(* PLC project desalination, Generated TextualNotationConverter 1.0 *)
(* stored: creationDateTime 2025-07-30T12:00:00, modificationDateTime 2025-01-30T12:00:00 *)

FUNCTION_BLOCK ANALOG_IN
  VAR_INPUT
    Name : STRING;
    Description : STRING;
    Raw_Signal : REAL;
    PV_High : REAL;
    PV_Low : REAL;
    Scaling_Slope : REAL;
    Scaling_Offset : REAL;
    Alarm_Enable : BOOL;
  END_VAR
  VAR_OUTPUT
    PV : REAL;
    High_Alarm : BOOL;
    Low_Alarm : BOOL;
    General_Fault : BOOL;
  END_VAR

            
          
END_FUNCTION_BLOCK

FUNCTION_BLOCK DIGITAL_IN
  VAR_INPUT
    Name : STRING;
    Description : STRING;
    DI_Raw : BOOL;
    DebounceTime : STRING;
    EnableAlarm : BOOL;
  END_VAR
  VAR_OUTPUT
    DI_Out : BOOL;
    Fault_State : BOOL;
  END_VAR

            
          
END_FUNCTION_BLOCK

FUNCTION_BLOCK PID_BASIC
  VAR_INPUT
    Name : STRING;
    Description : STRING;
    AUTO : BOOL;
    PV : REAL;
    SP : REAL;
    MV_MIN : REAL;
    MV_MAX : REAL;
    X0 : REAL;
    KP : REAL;
    TR : REAL;
    TD : REAL;
    PV_High : REAL;
    PV_Low : REAL;
    Deviation_Limit : REAL;
    Inhibit : BOOL;
  END_VAR
  VAR_OUTPUT
    PV_High_Alarm : BOOL;
    PV_Low_Alarm : BOOL;
    Deviation_Alarm : BOOL;
    XOUT : REAL;
  END_VAR

            
          
END_FUNCTION_BLOCK

FUNCTION_BLOCK VALVE_ELECTRIC
  VAR_INPUT
    Name : STRING;
    Description : STRING;
    Control_Signal : REAL;
    Manual_Mode : BOOL;
    Manual_Position : REAL;
    Open_Limit : REAL;
    Close_Limit : REAL;
    Timeout : STRING;
    Inhibit : BOOL;
  END_VAR
  VAR_OUTPUT
    Valve_Position : REAL;
    Feedback_Pos : REAL;
    Valve_Moving : BOOL;
    Position_Error : BOOL;
    Alarm : BOOL;
  END_VAR

            
          
END_FUNCTION_BLOCK

FUNCTION_BLOCK VALVE_ON_OFF
  VAR_INPUT
    Name : STRING;
    Description : STRING;
    Open_Cmd : BOOL;
    Close_Cmd : BOOL;
    Timeout : STRING;
    Inhibit : BOOL;
  END_VAR
  VAR_OUTPUT
    FB_Opened : BOOL;
    FB_Closed : BOOL;
    Valve_Open_Out : BOOL;
    Valve_Close_Out : BOOL;
    Alarm_Position_Error : BOOL;
    Alarm_General : BOOL;
  END_VAR

            
          
END_FUNCTION_BLOCK

PROGRAM Section2
  VAR
    AT_101_mA : REAL;
    AT_103_mA : REAL;
    FT_101_mA : REAL;
    FT_102_mA : REAL;
    LT_104_mA : REAL;
    LT_105_mA : REAL;
    XV_102_OpenLS_Raw : BOOL;
    XV_102_CloseLS_Raw : BOOL;
    SP_Seawater_Req : REAL;
    SP_Reservoir_Req : REAL;
    SP_Seawater_Clamped : REAL;
    SP_Reservoir_Clamped : REAL;
    FC_101_Auto_Cmd : BOOL;
    FC_102_Auto_Cmd : BOOL;
    FV_101_Manual_Mode : BOOL;
    FV_102_Manual_Mode : BOOL;
    FV_101_Manual_Position : REAL;
    FV_102_Manual_Position : REAL;
    FT_101_Flow_PV : REAL;
    FT_102_Flow_PV : REAL;
    FC_101_PID_Output : REAL;
    FC_102_PID_Output : REAL;
    FV_101_Valve_Position : REAL;
    FV_102_Valve_Position : REAL;
    AT_101_Quality_PV : REAL;
    AT_103_Quality_PV : REAL;
    LT_104_Level_PV : REAL;
    LT_105_Level_PV : REAL;
    WaterQuality_Alarm : BOOL;
    FV101_Inhibit : BOOL;
    FV102_Inhibit : BOOL;
  END_VAR
  VAR
    AT-101 : ANALOG_IN;
    AT-103 : ANALOG_IN;
    FC-101 : PID_BASIC;
    FC-102 : PID_BASIC;
    FT-101 : ANALOG_IN;
    FT-102 : ANALOG_IN;
    FV-101 : VALVE_ELECTRIC;
    FV-102 : VALVE_ELECTRIC;
    LT-104 : ANALOG_IN;
    LT-105 : ANALOG_IN;
    XV-102 : VALVE_ON_OFF;
    XV-102_OPEN_LS : DIGITAL_IN;
    XV-102_CLOSE_LS : DIGITAL_IN;
  END_VAR
  VAR  (* added by the conversion: wires and edge detectors of the diagram *)
    _OR1_OUT : BOOL;
    _OR2_OUT : BOOL;
    _OR3_OUT : BOOL;
  END_VAR

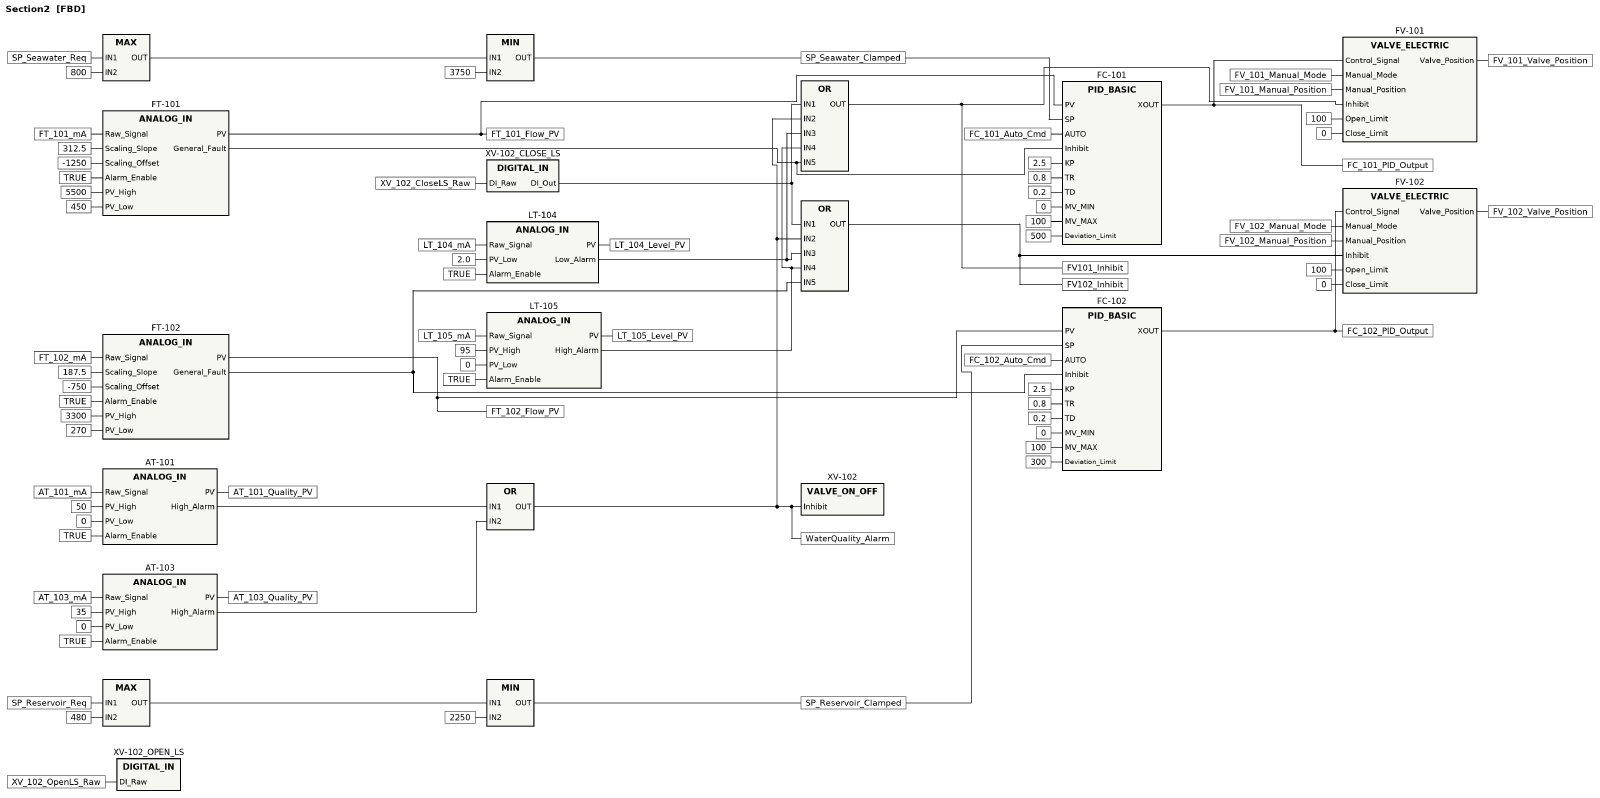
(* FBD diagram, written out as Structured Text *)
AT-101(Raw_Signal := AT_101_mA, PV_High := 50, PV_Low := 0, Alarm_Enable := TRUE);
AT_101_Quality_PV := AT-101.PV;
AT-103(Raw_Signal := AT_103_mA, PV_High := 35, PV_Low := 0, Alarm_Enable := TRUE);
AT_103_Quality_PV := AT-103.PV;
FT-101(Raw_Signal := FT_101_mA, Scaling_Slope := 312.5, Scaling_Offset := -1250, Alarm_Enable := TRUE, PV_High := 5500, PV_Low := 450);
FC-101(PV := FT-101.PV, SP := MIN(MAX(SP_Seawater_Req, 800), 3750), AUTO := FC_101_Auto_Cmd, Inhibit := FT-101.General_Fault, KP := 2.5, TR := 0.8, TD := 0.2, MV_MIN := 0, MV_MAX := 100, Deviation_Limit := 500);
FC_101_PID_Output := FC-101.XOUT;
FT-102(Raw_Signal := FT_102_mA, Scaling_Slope := 187.5, Scaling_Offset := -750, Alarm_Enable := TRUE, PV_High := 3300, PV_Low := 270);
FC-102(PV := FT-102.PV, SP := MIN(MAX(SP_Reservoir_Req, 480), 2250), AUTO := FC_102_Auto_Cmd, Inhibit := FT-102.General_Fault, KP := 2.5, TR := 0.8, TD := 0.2, MV_MIN := 0, MV_MAX := 100, Deviation_Limit := 300);
FC_102_PID_Output := FC-102.XOUT;
FT_101_Flow_PV := FT-101.PV;
FT_102_Flow_PV := FT-102.PV;
XV-102_CLOSE_LS(DI_Raw := XV_102_CloseLS_Raw);
_OR1_OUT := AT-101.High_Alarm OR AT-103.High_Alarm;
LT-104(Raw_Signal := LT_104_mA, PV_Low := 2.0, Alarm_Enable := TRUE);
LT-105(Raw_Signal := LT_105_mA, PV_High := 95, PV_Low := 0, Alarm_Enable := TRUE);
_OR2_OUT := XV-102_CLOSE_LS.DI_Out OR _OR1_OUT OR LT-104.Low_Alarm OR LT-105.High_Alarm OR FT-101.General_Fault;
FV101_Inhibit := _OR2_OUT;
_OR3_OUT := XV-102_CLOSE_LS.DI_Out OR _OR1_OUT OR LT-104.Low_Alarm OR LT-105.High_Alarm OR FT-102.General_Fault;
FV102_Inhibit := _OR3_OUT;
FV-101(Control_Signal := FC-101.XOUT, Manual_Mode := FV_101_Manual_Mode, Manual_Position := FV_101_Manual_Position, Inhibit := _OR2_OUT, Open_Limit := 100, Close_Limit := 0);
FV_101_Valve_Position := FV-101.Valve_Position;
FV-102(Control_Signal := FC-102.XOUT, Manual_Mode := FV_102_Manual_Mode, Manual_Position := FV_102_Manual_Position, Inhibit := _OR3_OUT, Open_Limit := 100, Close_Limit := 0);
FV_102_Valve_Position := FV-102.Valve_Position;
LT_104_Level_PV := LT-104.PV;
LT_105_Level_PV := LT-105.PV;
SP_Reservoir_Clamped := MIN(MAX(SP_Reservoir_Req, 480), 2250);
SP_Seawater_Clamped := MIN(MAX(SP_Seawater_Req, 800), 3750);
WaterQuality_Alarm := _OR1_OUT;
XV-102(Inhibit := _OR1_OUT);
XV-102_OPEN_LS(DI_Raw := XV_102_OpenLS_Raw);
END_PROGRAM

FUNCTION_BLOCK BOOL_IN
  VAR_INPUT
    Name : STRING;
    Description : STRING;
    Bool_In : BOOL;
    Alarm_OnTrue : BOOL;
    Alarm_OnFalse : BOOL;
    Latch_Enable : BOOL;
    Reset_Latch : BOOL;
  END_VAR
  VAR_OUTPUT
    Bool_Out : BOOL;
    Alarm_Active : BOOL;
    Latched_Status : BOOL;
  END_VAR

            
          
END_FUNCTION_BLOCK

FUNCTION_BLOCK DUTY_STANDBY
  VAR_INPUT
    Name : STRING;
    Description : STRING;
    Enable : BOOL;
    StartRequest : BOOL;
    AlternateEnable : BOOL;
    ForcePumpA : BOOL;
    ForcePumpB : BOOL;
    DutyElapsed : BOOL;
    MinRunElapsed : BOOL;
    SwitchoverDelayElapsed : BOOL;
    StartTimeoutElapsed : BOOL;
    PumpA_RunFB : BOOL;
    PumpB_RunFB : BOOL;
    PumpA_Fault : BOOL;
    PumpB_Fault : BOOL;
    Reset : BOOL;
    Inhibit : BOOL;
  END_VAR
  VAR_OUTPUT
    CmdPumpA : BOOL;
    CmdPumpB : BOOL;
    ActiveIsA : BOOL;
    SwitchedDueToDuty : BOOL;
    SwitchedDueToFailure : BOOL;
    Alarm_FailedStart_A : BOOL;
    Alarm_FailedStart_B : BOOL;
    Alarm_NoAvailablePump : BOOL;
  END_VAR

            
          
END_FUNCTION_BLOCK

FUNCTION_BLOCK MOTOR_2SPD
  VAR_INPUT
    Name : STRING;
    Description : STRING;
    Start_Cmd : BOOL;
    Stop_Cmd : BOOL;
    Speed_High_Cmd : BOOL;
    Speed_Low_Cmd : BOOL;
    Inhibit : BOOL;
  END_VAR
  VAR_OUTPUT
    Motor_Start_Out : BOOL;
    FB_Running : BOOL;
    FB_Trip : BOOL;
    FB_HighSpeed : BOOL;
    FB_LowSpeed : BOOL;
    Alarm_Speed_Error : BOOL;
  END_VAR

            
          
END_FUNCTION_BLOCK

FUNCTION_BLOCK MOTOR_ON_OFF
  VAR_INPUT
    Name : STRING;
    Description : STRING;
    Start_Cmd : BOOL;
    Stop_Cmd : BOOL;
    Start_Delay : STRING;
    MinRunTime : STRING;
    Inhibit : BOOL;
  END_VAR
  VAR_OUTPUT
    Motor_Start_Out : BOOL;
    FB_Running : BOOL;
    FB_Trip : BOOL;
    Alarm_Start_Fail : BOOL;
    Alarm_Stop_Fail : BOOL;
  END_VAR

            
          
END_FUNCTION_BLOCK

FUNCTION_BLOCK MOTOR_VSD
  VAR_INPUT
    Name : STRING;
    Description : STRING;
    Start_Cmd : BOOL;
    Stop_Cmd : BOOL;
    Speed_SP : REAL;
    Accel_Ramp : STRING;
    Decel_Ramp : STRING;
    Inhibit : BOOL;
  END_VAR
  VAR_OUTPUT
    Speed_Out : REAL;
    FB_Running : BOOL;
    FB_Fault : BOOL;
    FB_Ready : BOOL;
    FB_ActualSpeed : REAL;
    Alarm_Speed_Deviation : BOOL;
    Alarm_Comm_Fail : BOOL;
  END_VAR

            
          
END_FUNCTION_BLOCK

FUNCTION_BLOCK RATIO_CONTROL
  VAR_INPUT
    Name : STRING;
    Description : STRING;
    Auto : BOOL;
    PrimaryPV : REAL;
    SecondaryPV : REAL;
    RatioSP : REAL;
    Bias : REAL;
    TrimKp : REAL;
    TrimTi : STRING;
    MV_MIN : REAL;
    MV_MAX : REAL;
    ManOut : REAL;
    Inhibit : BOOL;
  END_VAR
  VAR_OUTPUT
    SlaveSP : REAL;
    ActiveRatio : REAL;
    RatioErr : REAL;
  END_VAR

            
          
END_FUNCTION_BLOCK

FUNCTION_BLOCK SPLIT_RANGE
  VAR_INPUT
    Name : STRING;
    Description : STRING;
    IN : REAL;
    Split_Point : REAL;
    Output1_Start : REAL;
    Output1_End : REAL;
    Output2_Start : REAL;
    Output2_End : REAL;
  END_VAR
  VAR_OUTPUT
    OUT1 : REAL;
    OUT2 : REAL;
  END_VAR

            
          
END_FUNCTION_BLOCK

FUNCTION_BLOCK VOTING_ANALOG
  VAR_INPUT
    Name : STRING;
    Description : STRING;
    Input1 : REAL;
    Input2 : REAL;
    Input3 : REAL;
    Deviation_Limit : REAL;
    Voting_Scheme : STRING;
    EnableAlarm : BOOL;
    Inhibit : BOOL;
  END_VAR
  VAR_OUTPUT
    Voted_Output : REAL;
    Sensor1_Fault : BOOL;
    Sensor2_Fault : BOOL;
    Sensor3_Fault : BOOL;
    Alarm_Voting_Error : BOOL;
    Healthy_Sensors_Count : INT;
  END_VAR

            
          
END_FUNCTION_BLOCK

PROGRAM Section3
  VAR
    FT101_SupplyAirFlow_PV : REAL;
    FT102_ScreenAirFlow_PV : REAL;
    PT103_UpstreamPressure_PV : REAL;
    PT104_DownstreamPressure_PV : REAL;
    PIT105_CompressedAirPressure_PV : REAL;
    PIT106_CleaningSystemPressure_PV : REAL;
    PT108_SupplyPressure_PV : REAL;
    FFIC103_SlaveSetpoint_FT102Flow : REAL;
    FIC104_ValveCommand_Percent : REAL;
    FV105_ValvePosition_Percent : REAL;
    FV105_FeedbackPosition_Percent : REAL;
    SW_SCREEN_1_Status : BOOL;
    SW_SCREEN_2_Status : BOOL;
    SW_SCREEN_3_Status : BOOL;
    SW_SCREEN_4_Status : BOOL;
    SW_SCREEN_5_Status : BOOL;
    SW_SCREEN_6_Status : BOOL;
    RES_SCREEN_1_Status : BOOL;
    RES_SCREEN_2_Status : BOOL;
    RES_SCREEN_3_Status : BOOL;
    RES_SCREEN_4_Status : BOOL;
  END_VAR
  VAR
    FFIC-103 : RATIO_CONTROL;
    FIC-104 : PID_BASIC;
    FV-105 : VALVE_ELECTRIC;
    FT-101 : ANALOG_IN;
    FT-102 : ANALOG_IN;
    PIT-105 : ANALOG_IN;
    PIT-106 : ANALOG_IN;
    PT-103 : ANALOG_IN;
    PT-104 : ANALOG_IN;
    PT-108 : ANALOG_IN;
    SW-SCREEN-1 : BOOL_IN;
    SW-SCREEN-2 : BOOL_IN;
    SW-SCREEN-3 : BOOL_IN;
    SW-SCREEN-4 : BOOL_IN;
    SW-SCREEN-5 : BOOL_IN;
    SW-SCREEN-6 : BOOL_IN;
    RES-SCREEN-1 : BOOL_IN;
    RES-SCREEN-2 : BOOL_IN;
    RES-SCREEN-3 : BOOL_IN;
    RES-SCREEN-4 : BOOL_IN;
  END_VAR
  VAR  (* added by the conversion: wires and edge detectors of the diagram *)
    _OR94_OUT : BOOL;
  END_VAR

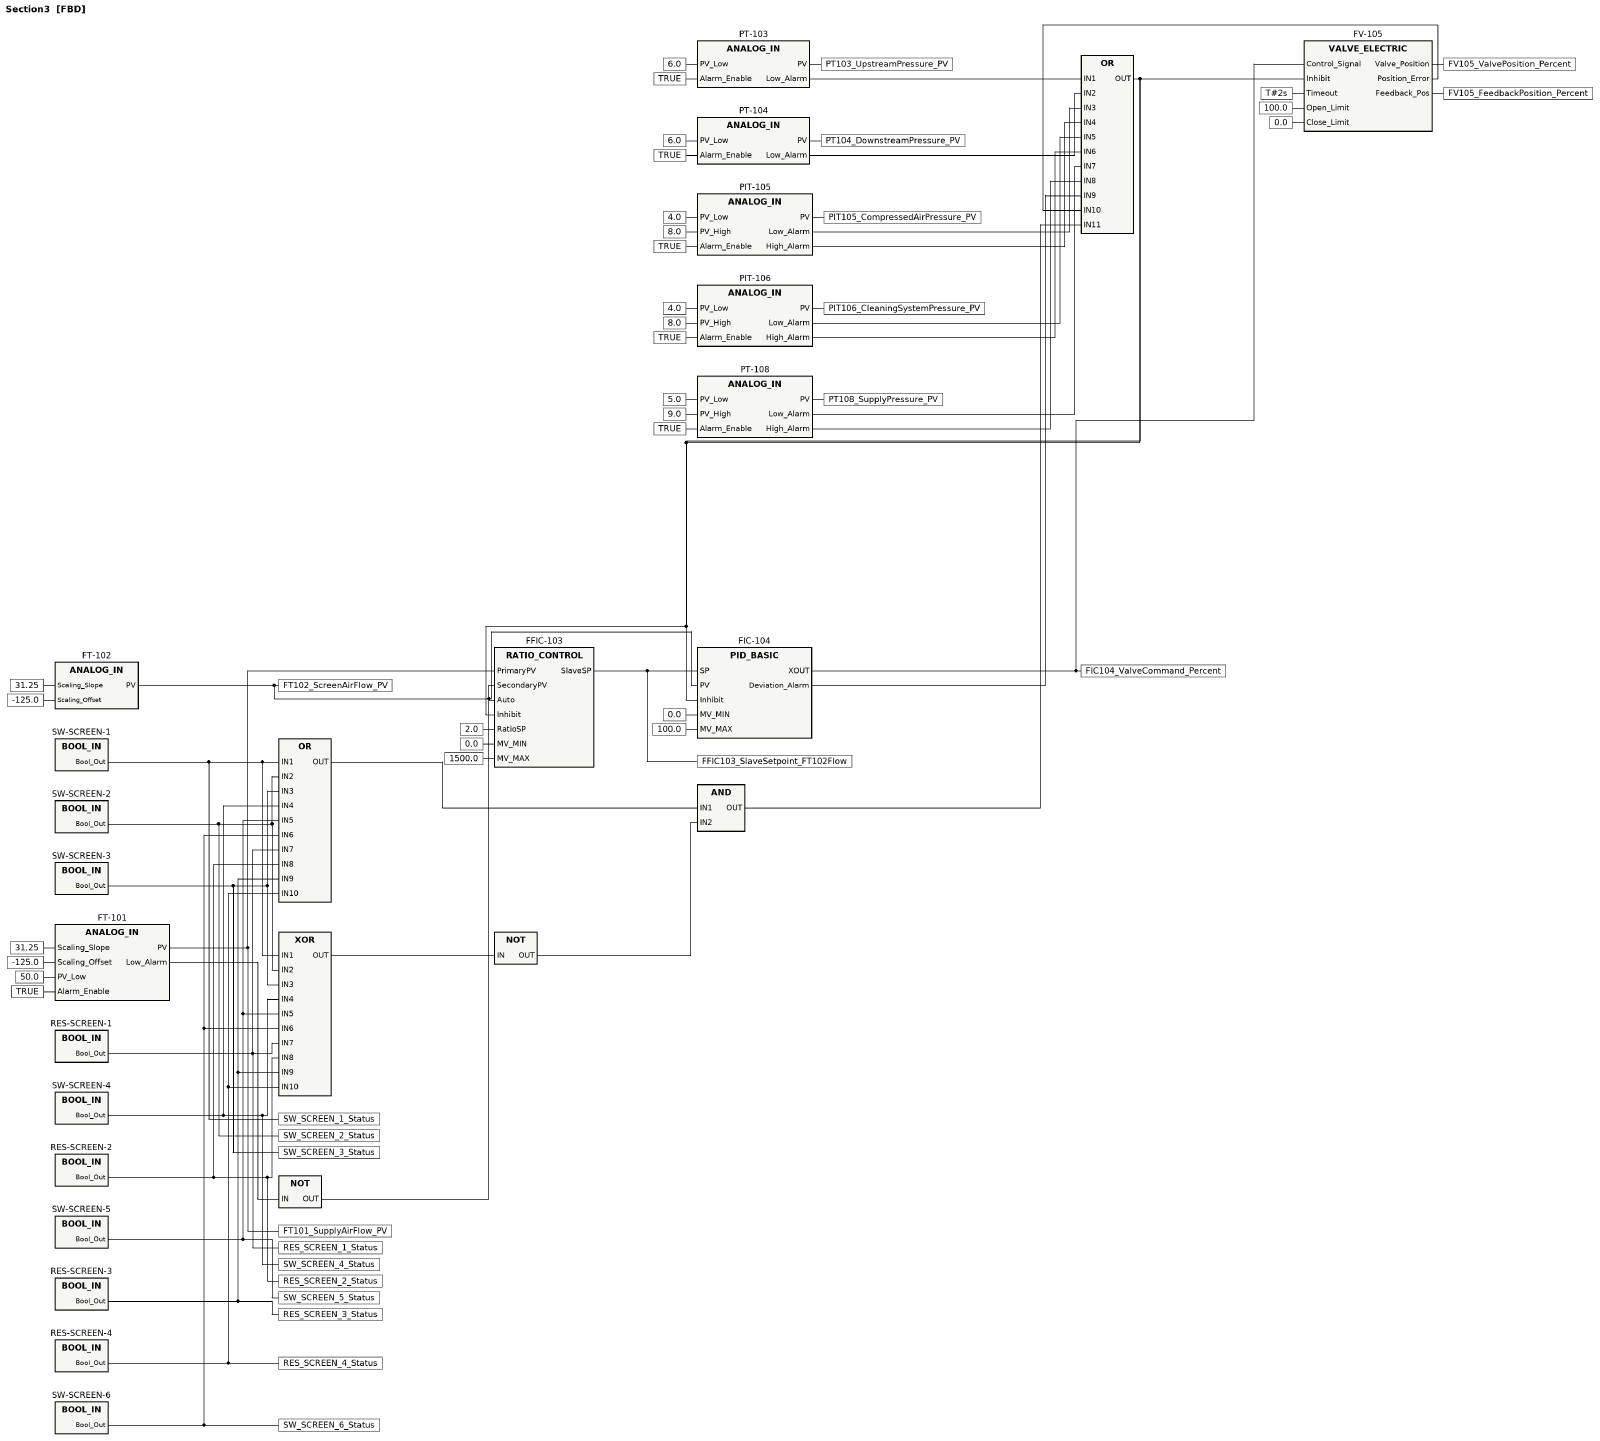
(* FBD diagram, written out as Structured Text *)
FT-101(Scaling_Slope := 31.25, Scaling_Offset := -125.0, PV_Low := 50.0, Alarm_Enable := TRUE);
FT-102(Scaling_Slope := 31.25, Scaling_Offset := -125.0);
PT-103(PV_Low := 6.0, Alarm_Enable := TRUE);
PT-104(PV_Low := 6.0, Alarm_Enable := TRUE);
PIT-105(PV_Low := 4.0, PV_High := 8.0, Alarm_Enable := TRUE);
PIT-106(PV_Low := 4.0, PV_High := 8.0, Alarm_Enable := TRUE);
PT-108(PV_Low := 5.0, PV_High := 9.0, Alarm_Enable := TRUE);
FIC-104(SP := FFIC-103.SlaveSP, PV := FT-102.PV, Inhibit := _OR94_OUT, MV_MIN := 0.0, MV_MAX := 100.0);
FV-105(Control_Signal := FIC-104.XOUT, Inhibit := _OR94_OUT, Timeout := T#2s, Open_Limit := 100.0, Close_Limit := 0.0);
SW-SCREEN-1();
SW-SCREEN-2();
SW-SCREEN-3();
SW-SCREEN-4();
SW-SCREEN-5();
SW-SCREEN-6();
RES-SCREEN-1();
RES-SCREEN-2();
RES-SCREEN-3();
RES-SCREEN-4();
_OR94_OUT := PT-103.Low_Alarm OR PT-104.Low_Alarm OR PIT-105.Low_Alarm OR PIT-105.High_Alarm OR PIT-106.Low_Alarm OR PIT-106.High_Alarm OR PT-108.Low_Alarm OR PT-108.High_Alarm OR FIC-104.Deviation_Alarm OR FV-105.Position_Error OR (SW-SCREEN-1.Bool_Out OR SW-SCREEN-2.Bool_Out OR SW-SCREEN-3.Bool_Out OR SW-SCREEN-4.Bool_Out OR SW-SCREEN-5.Bool_Out OR SW-SCREEN-6.Bool_Out OR RES-SCREEN-1.Bool_Out OR RES-SCREEN-2.Bool_Out OR RES-SCREEN-3.Bool_Out OR RES-SCREEN-4.Bool_Out) AND NOT (SW-SCREEN-1.Bool_Out XOR SW-SCREEN-2.Bool_Out XOR SW-SCREEN-3.Bool_Out XOR SW-SCREEN-4.Bool_Out XOR SW-SCREEN-5.Bool_Out XOR SW-SCREEN-6.Bool_Out XOR RES-SCREEN-1.Bool_Out XOR RES-SCREEN-2.Bool_Out XOR RES-SCREEN-3.Bool_Out XOR RES-SCREEN-4.Bool_Out);
FFIC-103(PrimaryPV := FT-101.PV, SecondaryPV := FT-102.PV, Auto := NOT FT-101.Low_Alarm, Inhibit := _OR94_OUT, RatioSP := 2.0, MV_MIN := 0.0, MV_MAX := 1500.0);
FFIC103_SlaveSetpoint_FT102Flow := FFIC-103.SlaveSP;
FIC104_ValveCommand_Percent := FIC-104.XOUT;
FT101_SupplyAirFlow_PV := FT-101.PV;
FT102_ScreenAirFlow_PV := FT-102.PV;
FV105_FeedbackPosition_Percent := FV-105.Feedback_Pos;
FV105_ValvePosition_Percent := FV-105.Valve_Position;
PIT105_CompressedAirPressure_PV := PIT-105.PV;
PIT106_CleaningSystemPressure_PV := PIT-106.PV;
PT103_UpstreamPressure_PV := PT-103.PV;
PT104_DownstreamPressure_PV := PT-104.PV;
PT108_SupplyPressure_PV := PT-108.PV;
RES_SCREEN_1_Status := RES-SCREEN-1.Bool_Out;
RES_SCREEN_2_Status := RES-SCREEN-2.Bool_Out;
RES_SCREEN_3_Status := RES-SCREEN-3.Bool_Out;
RES_SCREEN_4_Status := RES-SCREEN-4.Bool_Out;
SW_SCREEN_1_Status := SW-SCREEN-1.Bool_Out;
SW_SCREEN_2_Status := SW-SCREEN-2.Bool_Out;
SW_SCREEN_3_Status := SW-SCREEN-3.Bool_Out;
SW_SCREEN_4_Status := SW-SCREEN-4.Bool_Out;
SW_SCREEN_5_Status := SW-SCREEN-5.Bool_Out;
SW_SCREEN_6_Status := SW-SCREEN-6.Bool_Out;
END_PROGRAM

PROGRAM Section4
  VAR
    FT101_FlowRate_PV_m3h : REAL;
    LT101_SumpLevel_PV_m : REAL;
    FIC101_MV_Percent_ToVFD : REAL;
    FIC101_SP_m3h : REAL;
    ALM_FlowDeviation : BOOL;
    ALM_SumpLevelCritical : BOOL;
    M103A_EnableAlarm : BOOL;
    M103B_EnableAlarm : BOOL;
    M103C_EnableAlarm : BOOL;
    M103D_EnableAlarm : BOOL;
    SumpHighThreshold_m : REAL;
    SumpCriticalLowThreshold_m : REAL;
    SumpCriticalHighThreshold_m : REAL;
    FALSE_CONST : BOOL;
  END_VAR
  VAR
    FT-101 : ANALOG_IN;
    LT-101 : ANALOG_IN;
    FIC-101 : PID_BASIC;
    VFD-101A : MOTOR_VSD;
    VFD-101B : MOTOR_VSD;
    VFD-101C : MOTOR_VSD;
    VFD-101D : MOTOR_VSD;
    SPUMP-201A : MOTOR_ON_OFF;
    SPUMP-201B : MOTOR_ON_OFF;
    M103A : DIGITAL_IN;
    M103B : DIGITAL_IN;
    M103C : DIGITAL_IN;
    M103D : DIGITAL_IN;
    LEAK-101A : BOOL_IN;
    LEAK-101B : BOOL_IN;
    LEAK-101C : BOOL_IN;
    LEAK-101D : BOOL_IN;
    FlowDeviation_TON : TON;
  END_VAR
  VAR  (* added by the conversion: wires and edge detectors of the diagram *)
    _OR167_OUT : BOOL;
    _OR175_OUT : BOOL;
    _GT172_OUT : BOOL;
    _OR176_OUT : BOOL;
  END_VAR

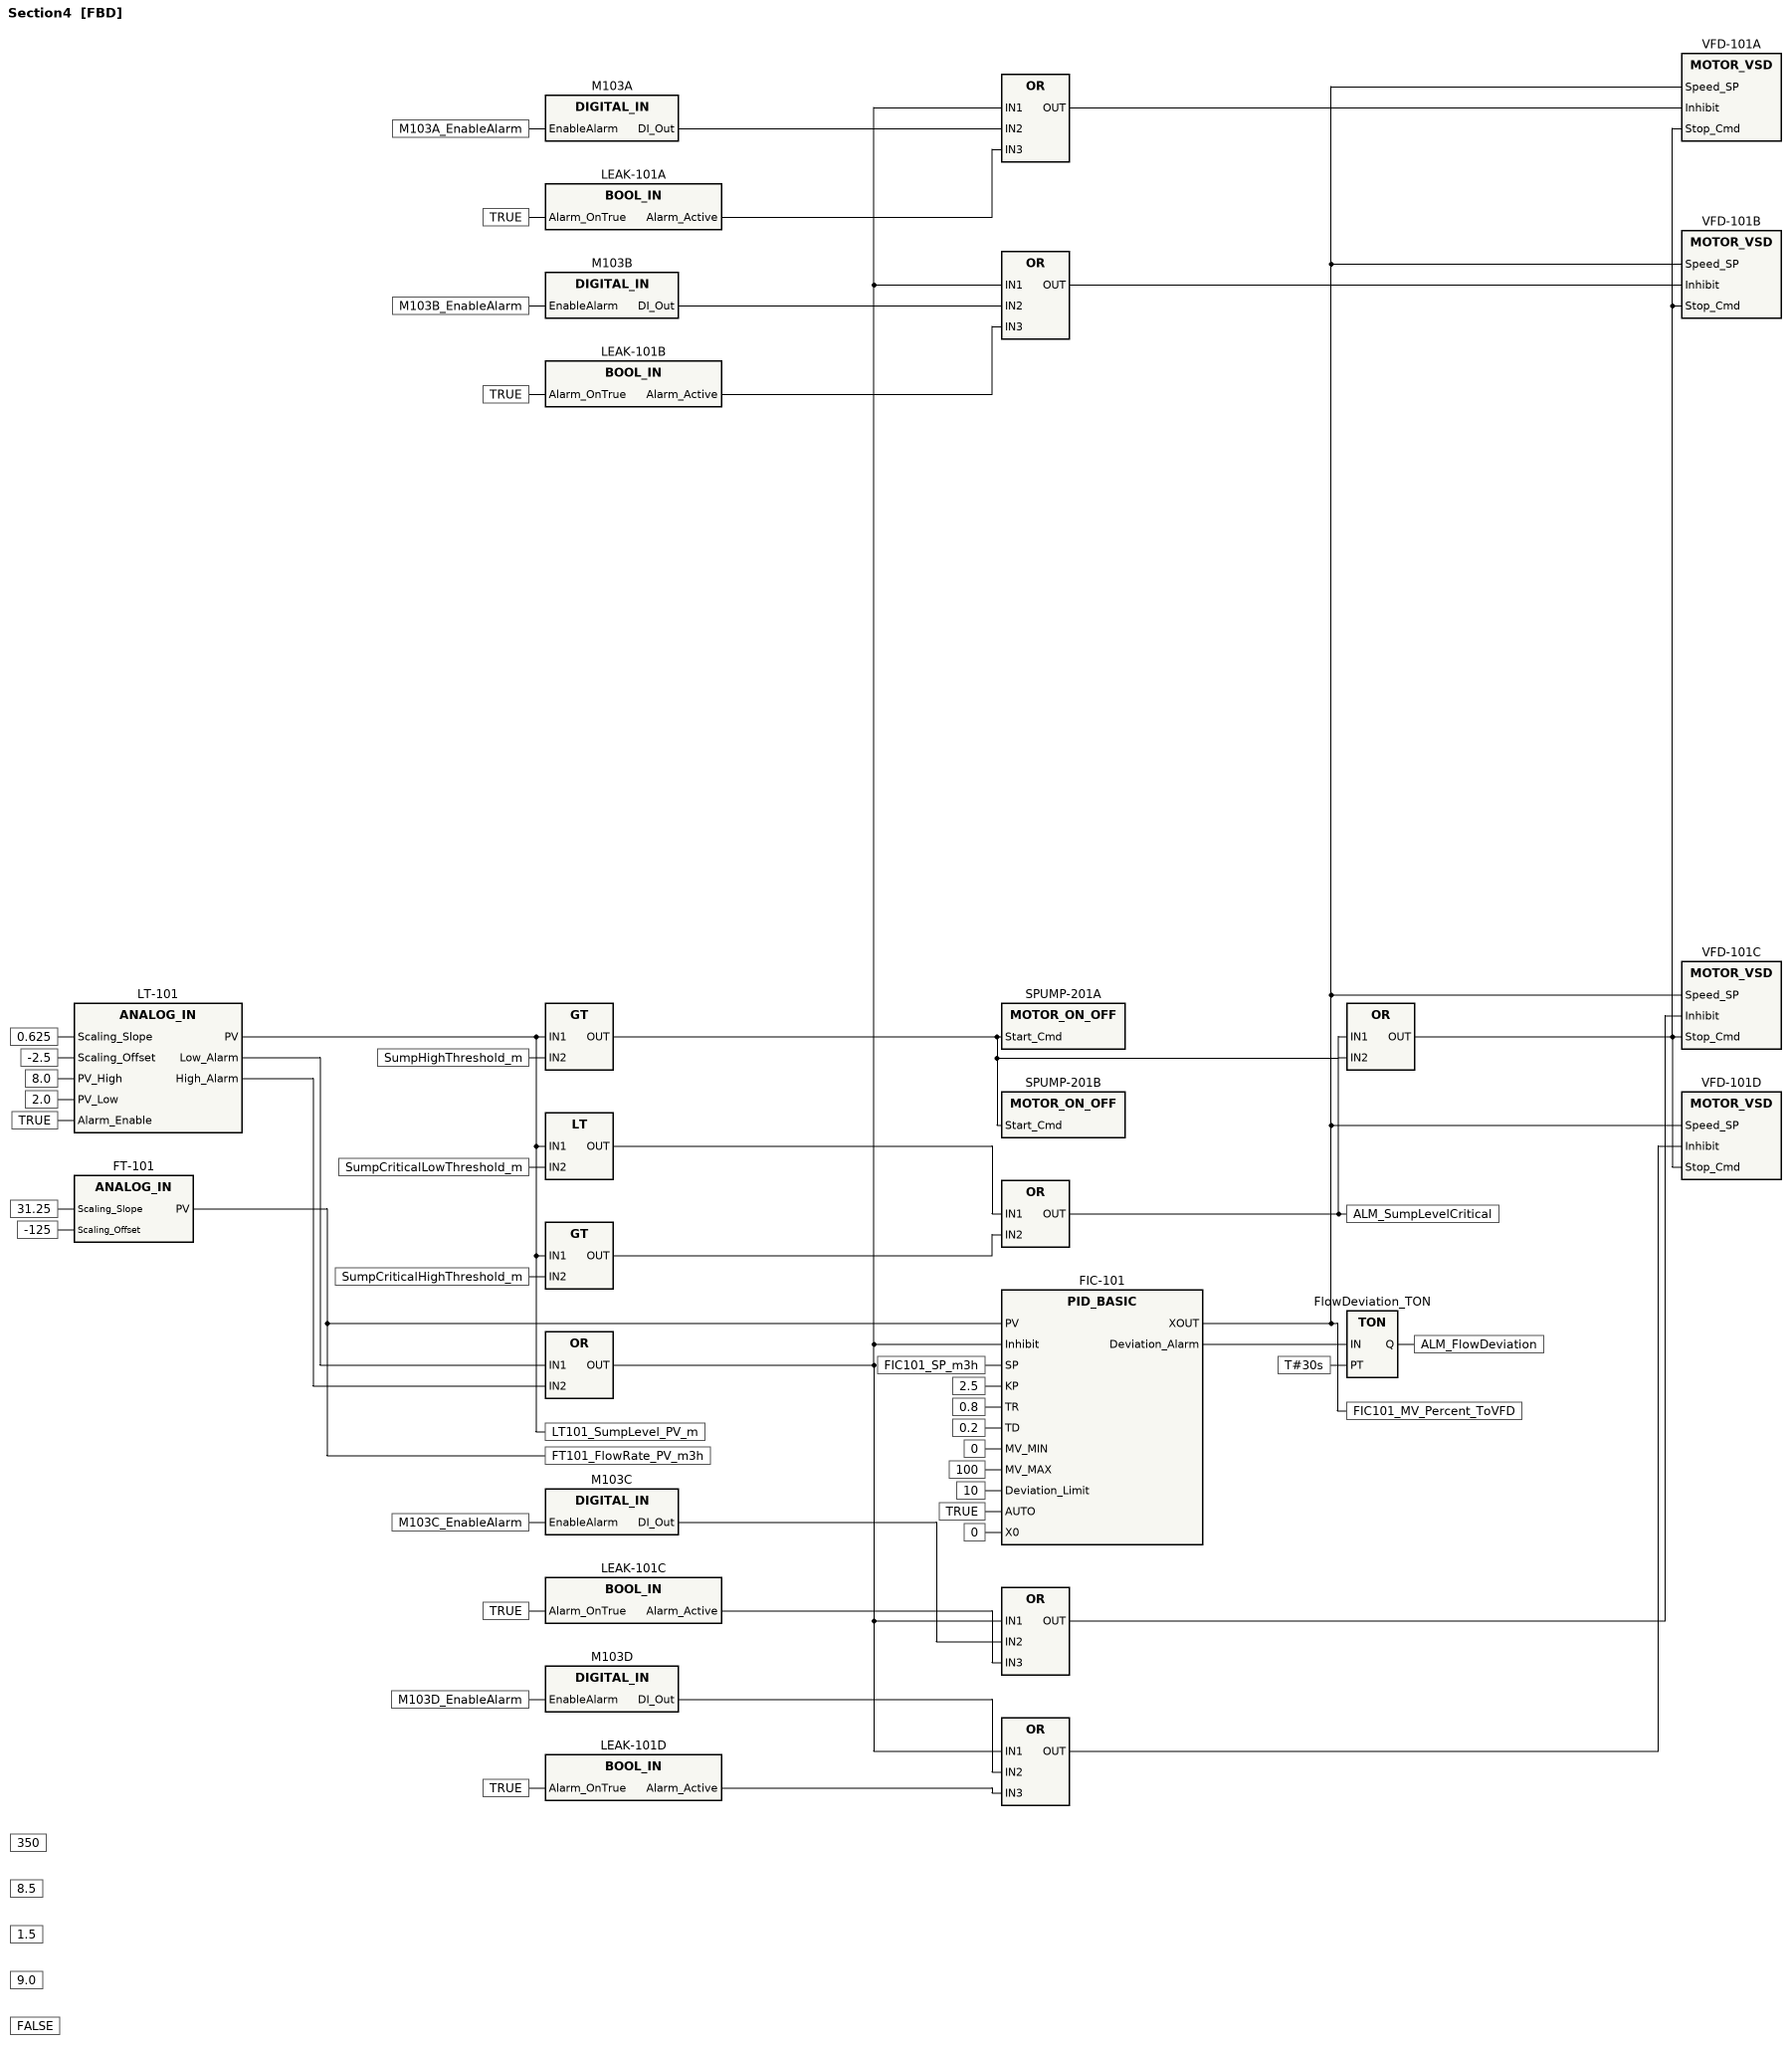
(* FBD diagram, written out as Structured Text *)
FT-101(Scaling_Slope := 31.25, Scaling_Offset := -125);
LT-101(Scaling_Slope := 0.625, Scaling_Offset := -2.5, PV_High := 8.0, PV_Low := 2.0, Alarm_Enable := TRUE);
_OR167_OUT := LT-101.Low_Alarm OR LT-101.High_Alarm;
FIC-101(PV := FT-101.PV, Inhibit := _OR167_OUT, SP := FIC101_SP_m3h, KP := 2.5, TR := 0.8, TD := 0.2, MV_MIN := 0, MV_MAX := 100, Deviation_Limit := 10, AUTO := TRUE, X0 := 0);
FlowDeviation_TON(IN := FIC-101.Deviation_Alarm, PT := T#30s);
ALM_FlowDeviation := FlowDeviation_TON.Q;
_OR175_OUT := LT-101.PV < SumpCriticalLowThreshold_m OR LT-101.PV > SumpCriticalHighThreshold_m;
ALM_SumpLevelCritical := _OR175_OUT;
FIC101_MV_Percent_ToVFD := FIC-101.XOUT;
FT101_FlowRate_PV_m3h := FT-101.PV;
LT101_SumpLevel_PV_m := LT-101.PV;
M103A(EnableAlarm := M103A_EnableAlarm);
LEAK-101A(Alarm_OnTrue := TRUE);
M103B(EnableAlarm := M103B_EnableAlarm);
LEAK-101B(Alarm_OnTrue := TRUE);
M103C(EnableAlarm := M103C_EnableAlarm);
LEAK-101C(Alarm_OnTrue := TRUE);
M103D(EnableAlarm := M103D_EnableAlarm);
LEAK-101D(Alarm_OnTrue := TRUE);
_GT172_OUT := LT-101.PV > SumpHighThreshold_m;
_OR176_OUT := _GT172_OUT OR _OR175_OUT;
VFD-101A(Speed_SP := FIC-101.XOUT, Inhibit := _OR167_OUT OR M103A.DI_Out OR LEAK-101A.Alarm_Active, Stop_Cmd := _OR176_OUT);
VFD-101B(Speed_SP := FIC-101.XOUT, Inhibit := _OR167_OUT OR M103B.DI_Out OR LEAK-101B.Alarm_Active, Stop_Cmd := _OR176_OUT);
VFD-101C(Speed_SP := FIC-101.XOUT, Inhibit := _OR167_OUT OR M103C.DI_Out OR LEAK-101C.Alarm_Active, Stop_Cmd := _OR176_OUT);
VFD-101D(Speed_SP := FIC-101.XOUT, Inhibit := _OR167_OUT OR M103D.DI_Out OR LEAK-101D.Alarm_Active, Stop_Cmd := _OR176_OUT);
SPUMP-201A(Start_Cmd := _GT172_OUT);
SPUMP-201B(Start_Cmd := _GT172_OUT);
(* drawn but not wired to any output: 350, 8.5, 1.5, 9.0, FALSE *)
END_PROGRAM

PROGRAM Section5
  VAR
    CHLOR-PUMP-301AB_Stroke_CMD : REAL;
  END_VAR
  VAR
    ANK-301 : BOOL_IN;
    FAH-301 : DIGITAL_IN;
    FAL-301 : DIGITAL_IN;
    FIC-301 : PID_BASIC;
    FT-301 : ANALOG_IN;
    FV-301 : VALVE_ELECTRIC;
    LAL-301 : DIGITAL_IN;
    LT-301 : ANALOG_IN;
    PAH-103 : DIGITAL_IN;
    PFA-301 : DIGITAL_IN;
    TAH-101 : DIGITAL_IN;
    UMP-301A : MOTOR_VSD;
    UMP-301B : MOTOR_VSD;
    XV-107 : VALVE_ON_OFF;
  END_VAR
  VAR  (* added by the conversion: wires and edge detectors of the diagram *)
    _OR238_OUT : BOOL;
    _OR241_OUT : BOOL;
  END_VAR

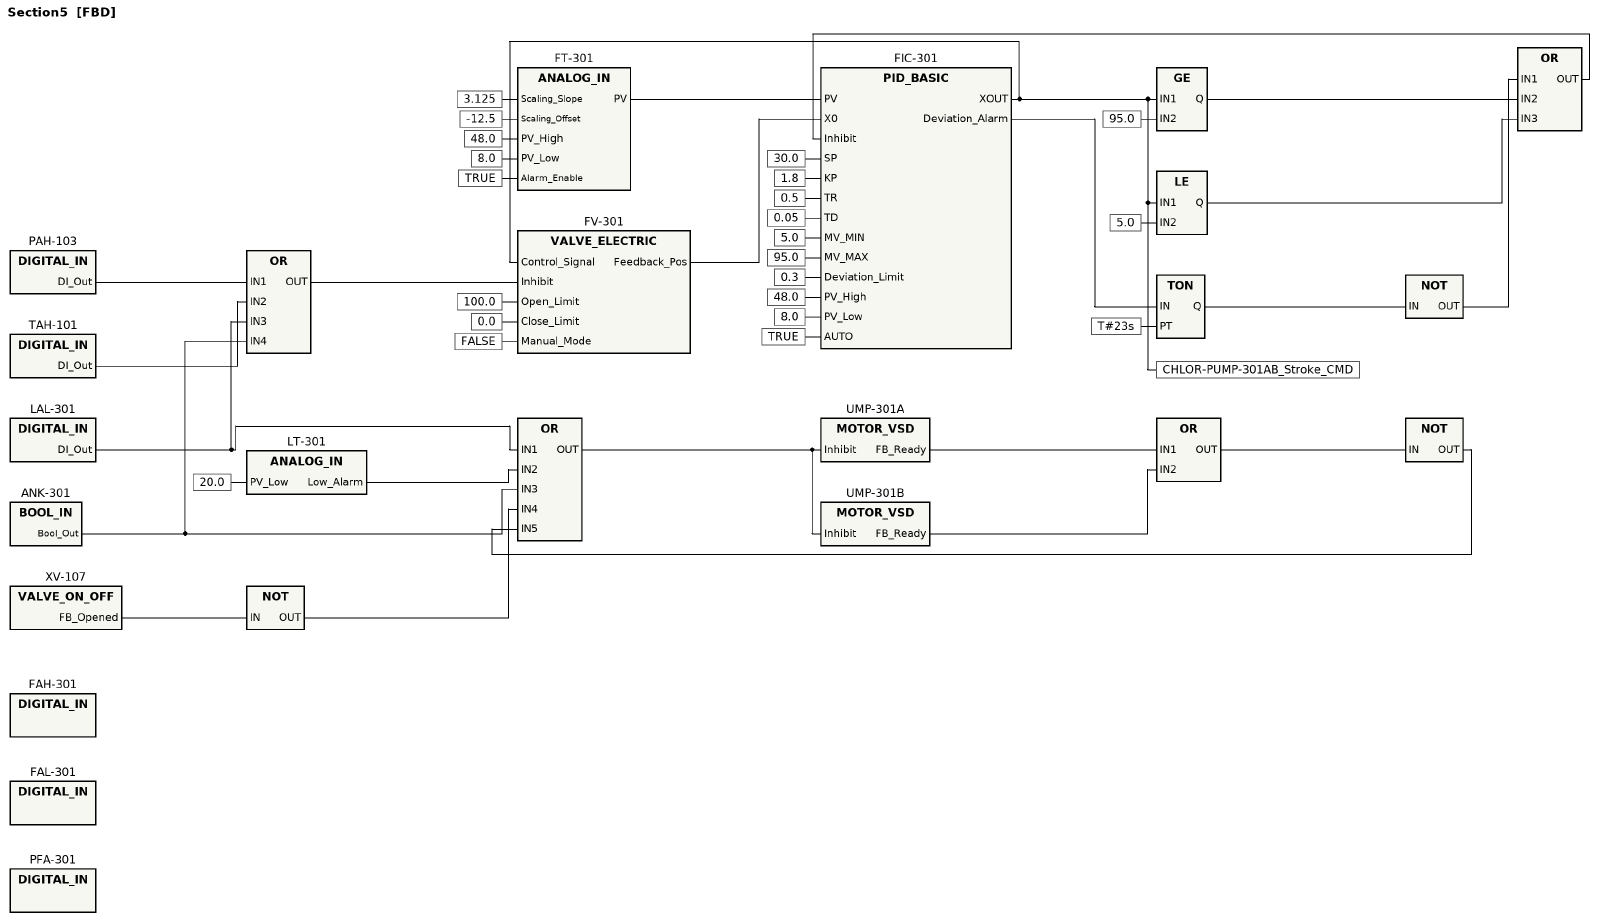
(* FBD diagram, written out as Structured Text *)
FT-301(Scaling_Slope := 3.125, Scaling_Offset := -12.5, PV_High := 48.0, PV_Low := 8.0, Alarm_Enable := TRUE);
PAH-103();
TAH-101();
LAL-301();
ANK-301();
FV-301(Control_Signal := FIC-301.XOUT, Inhibit := PAH-103.DI_Out OR TAH-101.DI_Out OR LAL-301.DI_Out OR ANK-301.Bool_Out, Open_Limit := 100.0, Close_Limit := 0.0, Manual_Mode := FALSE);
FIC-301(PV := FT-301.PV, X0 := FV-301.Feedback_Pos, Inhibit := NOT TON(FIC-301.Deviation_Alarm, T#23s) OR FIC-301.XOUT >= 95.0 OR FIC-301.XOUT <= 5.0, SP := 30.0, KP := 1.8, TR := 0.5, TD := 0.05, MV_MIN := 5.0, MV_MAX := 95.0, Deviation_Limit := 0.3, PV_High := 48.0, PV_Low := 8.0, AUTO := TRUE);
CHLOR-PUMP-301AB_Stroke_CMD := FIC-301.XOUT;
LT-301(PV_Low := 20.0);
XV-107();
_OR241_OUT := LAL-301.DI_Out OR LT-301.Low_Alarm OR ANK-301.Bool_Out OR NOT XV-107.FB_Opened OR NOT _OR238_OUT;
UMP-301A(Inhibit := _OR241_OUT);
UMP-301B(Inhibit := _OR241_OUT);
_OR238_OUT := UMP-301A.FB_Ready OR UMP-301B.FB_Ready;
FAH-301();
FAL-301();
PFA-301();
END_PROGRAM

PROGRAM Section6
  VAR
    SamplingFlow_PV : REAL;
    FIT101_BypassFlow_PV : REAL;
    FIC104_SamplingFlow_SP : REAL;
    FIC104_ActiveSamplingToBypassRatio : REAL;
  END_VAR
  VAR
    FIT-101 : ANALOG_IN;
    AT-105 : BOOL_IN;
    FIC-104 : RATIO_CONTROL;
    FV-102 : VALVE_ELECTRIC;
    LV-103 : VALVE_ELECTRIC;
  END_VAR
  VAR  (* added by the conversion: wires and edge detectors of the diagram *)
    _OR282_OUT : BOOL;
  END_VAR

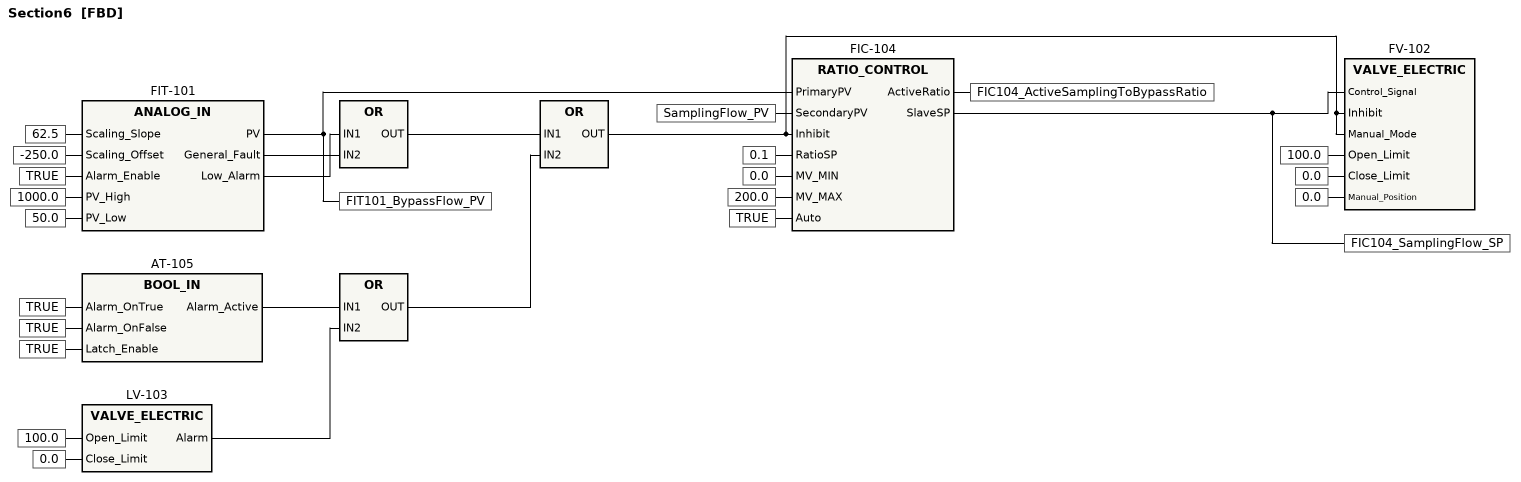
(* FBD diagram, written out as Structured Text *)
FIT-101(Scaling_Slope := 62.5, Scaling_Offset := -250.0, Alarm_Enable := TRUE, PV_High := 1000.0, PV_Low := 50.0);
AT-105(Alarm_OnTrue := TRUE, Alarm_OnFalse := TRUE, Latch_Enable := TRUE);
LV-103(Open_Limit := 100.0, Close_Limit := 0.0);
_OR282_OUT := FIT-101.Low_Alarm OR FIT-101.General_Fault OR AT-105.Alarm_Active OR LV-103.Alarm;
FIC-104(PrimaryPV := FIT-101.PV, SecondaryPV := SamplingFlow_PV, Inhibit := _OR282_OUT, RatioSP := 0.1, MV_MIN := 0.0, MV_MAX := 200.0, Auto := TRUE);
FIC104_ActiveSamplingToBypassRatio := FIC-104.ActiveRatio;
FIC104_SamplingFlow_SP := FIC-104.SlaveSP;
FIT101_BypassFlow_PV := FIT-101.PV;
FV-102(Control_Signal := FIC-104.SlaveSP, Inhibit := _OR282_OUT, Manual_Mode := _OR282_OUT, Open_Limit := 100.0, Close_Limit := 0.0, Manual_Position := 0.0);
END_PROGRAM

CONFIGURATION Config0
  RESOURCE Res0 ON PLC
    TASK task0(INTERVAL := T#20ms, PRIORITY := 0);
    PROGRAM instance0 WITH task0 : Section2;
    PROGRAM instance_1 WITH task0 : Section3;
    PROGRAM instance_2 WITH task0 : Section4;
    PROGRAM instance_3 WITH task0 : Section5;
    PROGRAM instance_4 WITH task0 : Section6;
  END_RESOURCE
END_CONFIGURATION
